Omron Sysmac Studio project distributing_station_with_timer_1.9_no_erorcheck (1) (Sysmac Studio 1.54.0.64019, StandardProject)

# Controller new_Controller_0: NJ301-1100 version 1.14
Units and slaves: Node1 : NX-ECC201 (E001); Unit 1 : NX-PC0020 (N1); Unit 2 : NX-ID5442 (N2); Unit 3 : NX-PC0010 (N3); Unit 4 : NX-PC0020 (N4); Unit 5 : NX-OD5121 (N5); Unit 6 : NX-PC0010 (N6); Power Supply : NJ-Px3001; CPU : NJ301-1100; 0 [Unit 0] : CJ1W-AD041-V1 (J01); 1 [Unit 1] : CJ1W-DA041 (J02); 2 : CJ1W-ID211 (J03); 3 : CJ1W-OC211 (J04)
Task PrimaryTask (priority 4, period or condition 1000): Program0

VAR_GLOBAL
    Station_1B2 : BOOL;  (* Ejection Cylinder Extended; at IOBus://rack#0/slot#2/Ch1_In/Ch1_In01; published *)
    Station_1B1 : BOOL;  (* Ejection Cylinder retracted; at IOBus://rack#0/slot#2/Ch1_In/Ch1_In02; published *)
    Station_2B1 : BOOL;  (* Workpiece gripped; at IOBus://rack#0/slot#2/Ch1_In/Ch1_In03; published *)
    Station_3S1 : BOOL;  (* arm_in_magazine; at IOBus://rack#0/slot#2/Ch1_In/Ch1_In04; published *)
    Station_3S2 : BOOL;  (* arm_in_downstream; at IOBus://rack#0/slot#2/Ch1_In/Ch1_In05; published *)
    Station_B4 : BOOL;  (* Magzine empty; at IOBus://rack#0/slot#2/Ch1_In/Ch1_In06; published *)
    Panel_S1 : BOOL;  (* start_button; at IOBus://rack#0/slot#2/Ch1_In/Ch1_In08; published *)
    Panel_S2 : BOOL;  (* stop_button; at IOBus://rack#0/slot#2/Ch1_In/Ch1_In09; published *)
    Panel_S4 : BOOL;  (* reset_button; at IOBus://rack#0/slot#2/Ch1_In/Ch1_In11; published *)
    Station_1Y1 : BOOL;  (* Magzine eject; at IOBus://rack#0/slot#3/Ch1_Out/Ch1_Out00; published *)
    Station_2Y1 : BOOL;  (* Vacuum on; at IOBus://rack#0/slot#3/Ch1_Out/Ch1_Out01; published *)
    Station_2Y2 : BOOL;  (* Ejector_Pulse_On; at IOBus://rack#0/slot#3/Ch1_Out/Ch1_Out02; published *)
    Station_3Y1 : BOOL;  (* arm_2_magazine; at IOBus://rack#0/slot#3/Ch1_Out/Ch1_Out03; published *)
    Station_3Y2 : BOOL;  (* arm_2_downstream; at IOBus://rack#0/slot#3/Ch1_Out/Ch1_Out04; published *)
    Station_H1 : BOOL;  (* start light; at IOBus://rack#0/slot#3/Ch1_Out/Ch1_Out08; published *)
    Station_H2 : BOOL;  (* reset light; at IOBus://rack#0/slot#3/Ch1_Out/Ch1_Out09; published *)
    Panel_H3 : BOOL;  (* Q1 light; at IOBus://rack#0/slot#3/Ch1_Out/Ch1_Out10; published *)
    Panel_H4 : BOOL;  (* Q2 light; at IOBus://rack#0/slot#3/Ch1_Out/Ch1_Out11; published *)
END_VAR

PROGRAM Program0
VAR
    FB_Panel_Distribution : FB_Panel;
    run_mode : BOOL;
    start_light : BOOL;
    reset_light : BOOL;
    pause_mode : BOOL;
    reset_mode : BOOL;
    T1_error_environment : BOOL;  (* t1 arm error *)
    error_mode : BOOL;
    T2_error_environment : BOOL;  (* t2 ejector error *)
    T1_to_end : BOOL;
    T1_to_home : BOOL;
    T1_at_home : BOOL;
    T1_at_end : BOOL;
    T2_to_end : BOOL;
    T2_to_home : BOOL;
    T2_at_home : BOOL;
    T2_at_end : BOOL;
    T2_Actuator_Env : T2_Actuator_No_RS_Controllable;
    T1_Actuator_Env : T1_Actuator_Controllable;
    Distrabution_Station_Logic_Env : Distrabuting_Station_Logic;
    manual_mode : BOOL;  (* empty boolean to control manual mode *)
    Dis_Logic_reset_light : BOOL;
    Dis_Logic_start_light : BOOL;
    Dis_Logic_empty_mag_light : BOOL;
    arm_to_end : BOOL;
    arm_to_home : BOOL;
    Dis_Logic_arm_to_end : BOOL;
    Dis_Logic_arm_to_home : BOOL;
    Dis_Logic_extend_mag_slide : BOOL;
    Dis_Logic_retract_mag_slide : BOOL;
END_VAR
VAR_EXTERNAL
    Station_3S1 : BOOL;
    Panel_S2 : BOOL;
    Station_3Y2 : BOOL;
    Station_3S2 : BOOL;
    Panel_S1 : BOOL;
    Station_3Y1 : BOOL;
    Station_H1 : BOOL;
    Station_H2 : BOOL;
    Panel_S4 : BOOL;
    Panel_H4 : BOOL;
    Station_1B1 : BOOL;
    Station_1B2 : BOOL;
    Station_1Y1 : BOOL;
    Station_2B1 : BOOL;
    Station_B4 : BOOL;
    Station_2Y1 : BOOL;
    Station_2Y2 : BOOL;
END_VAR

(* Section Section0: ladder, written here as Structured Text *)

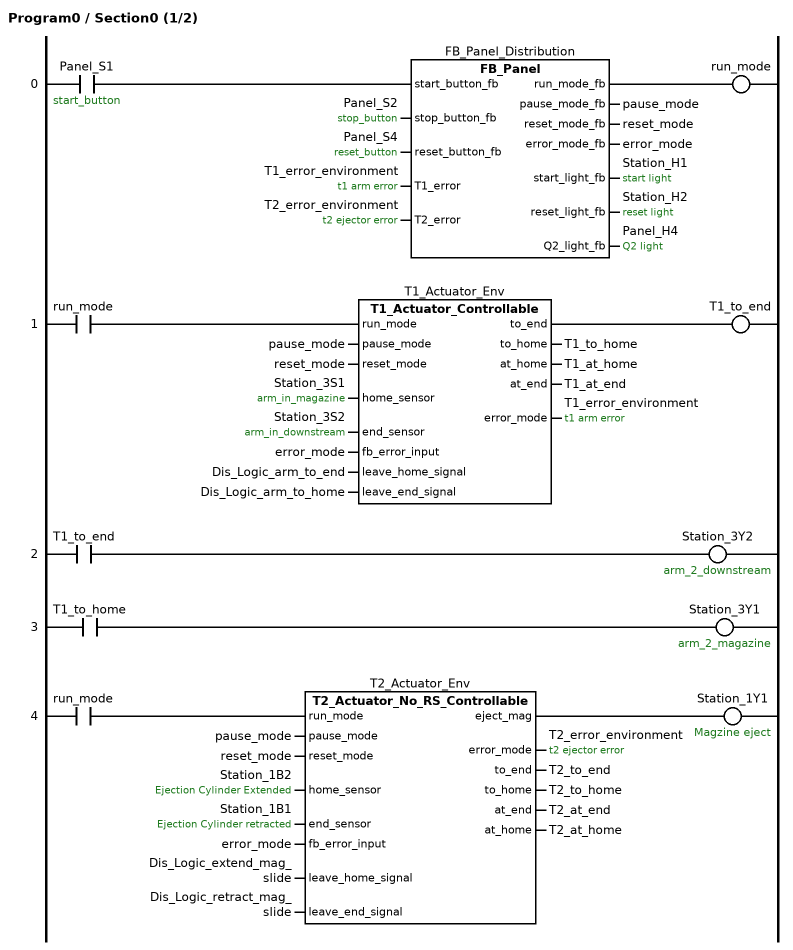
(* Rung 0 *)
FB_Panel_Distribution(start_button_fb := Panel_S1, stop_button_fb := Panel_S2, reset_button_fb := Panel_S4, T1_error := T1_error_environment, T2_error := T2_error_environment, pause_mode_fb => pause_mode, reset_mode_fb => reset_mode, error_mode_fb => error_mode, start_light_fb => Station_H1, reset_light_fb => Station_H2, Q2_light_fb => Panel_H4);
run_mode := FB_Panel_Distribution.run_mode_fb;
(* Rung 1 *)
T1_Actuator_Env(run_mode := run_mode, pause_mode := pause_mode, reset_mode := reset_mode, home_sensor := Station_3S1, end_sensor := Station_3S2, fb_error_input := error_mode, leave_home_signal := Dis_Logic_arm_to_end, leave_end_signal := Dis_Logic_arm_to_home, to_home => T1_to_home, at_home => T1_at_home, at_end => T1_at_end, error_mode => T1_error_environment);
T1_to_end := T1_Actuator_Env.to_end;
(* Rung 2 *)
Station_3Y2 := T1_to_end;
(* Rung 3 *)
Station_3Y1 := T1_to_home;
(* Rung 4 *)
T2_Actuator_Env(run_mode := run_mode, pause_mode := pause_mode, reset_mode := reset_mode, home_sensor := Station_1B2, end_sensor := Station_1B1, fb_error_input := error_mode, leave_home_signal := Dis_Logic_extend_mag_slide, leave_end_signal := Dis_Logic_retract_mag_slide, error_mode => T2_error_environment, to_end => T2_to_end, to_home => T2_to_home, at_end => T2_at_end, at_home => T2_at_home);
Station_1Y1 := T2_Actuator_Env.eject_mag;

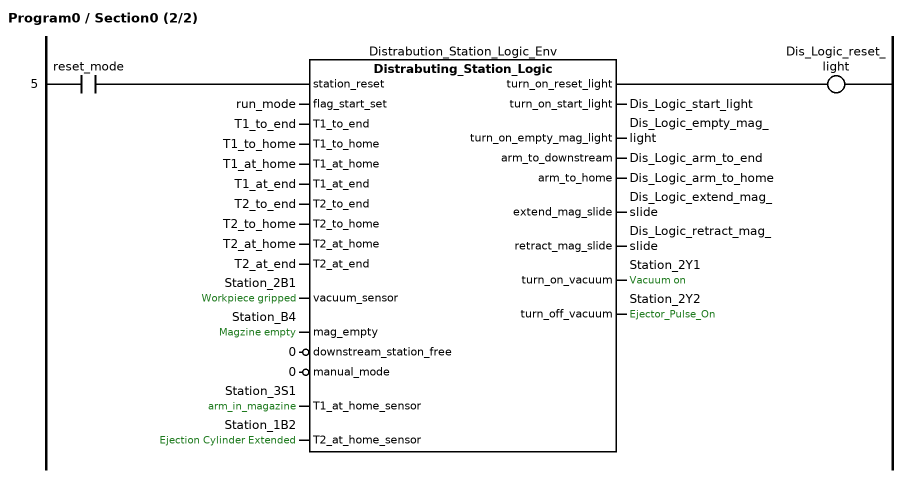
(* Rung 5 *)
Distrabution_Station_Logic_Env(station_reset := reset_mode, flag_start_set := run_mode, T1_to_end := T1_to_end, T1_to_home := T1_to_home, T1_at_home := T1_at_home, T1_at_end := T1_at_end, T2_to_end := T2_to_end, T2_to_home := T2_to_home, T2_at_home := T2_at_home, T2_at_end := T2_at_end, vacuum_sensor := Station_2B1, mag_empty := Station_B4, downstream_station_free := NOT 0, manual_mode := NOT 0, T1_at_home_sensor := Station_3S1, T2_at_home_sensor := Station_1B2, turn_on_start_light => Dis_Logic_start_light, turn_on_empty_mag_light => Dis_Logic_empty_mag_light, arm_to_downstream => Dis_Logic_arm_to_end, arm_to_home => Dis_Logic_arm_to_home, extend_mag_slide => Dis_Logic_extend_mag_slide, retract_mag_slide => Dis_Logic_retract_mag_slide, turn_on_vacuum => Station_2Y1, turn_off_vacuum => Station_2Y2);
Dis_Logic_reset_light := Distrabution_Station_Logic_Env.turn_on_reset_light;
END_PROGRAM

FUNCTION_BLOCK FB_Panel
VAR
    RS_run_mode : RS;
    RS_reset_mode : RS;
    RS_run_mode_reset : BOOL;  (* reset run mode RS *)
END_VAR
VAR_OUTPUT
    run_mode_fb : BOOL;
    pause_mode_fb : BOOL;
    reset_mode_fb : BOOL;
    error_mode_fb : BOOL;
END_VAR
VAR_INPUT
    start_button_fb : BOOL;
    stop_button_fb : BOOL;
    reset_button_fb : BOOL;
    T1_error : BOOL;  (* arm error mode input *)
    T2_error : BOOL;  (* ejector cylinder error mode input *)
END_VAR
VAR_OUTPUT
    start_light_fb : BOOL;
    reset_light_fb : BOOL;
    Q2_light_fb : BOOL;
END_VAR
(* ladder, written here as Structured Text *)

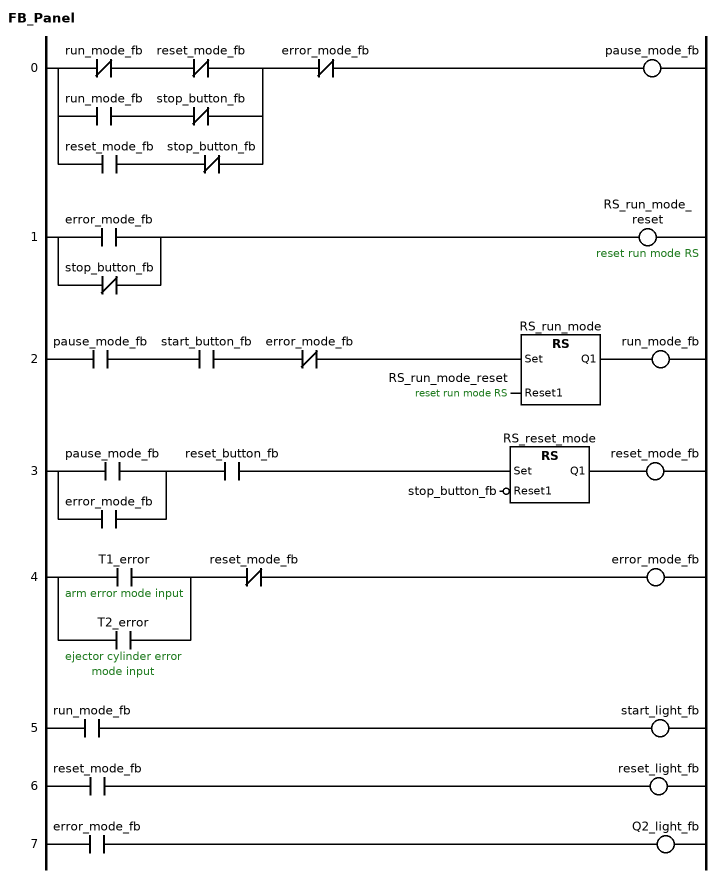
(* Rung 0 *)
pause_mode_fb := ((NOT run_mode_fb AND NOT reset_mode_fb) OR (run_mode_fb AND NOT stop_button_fb) OR (reset_mode_fb AND NOT stop_button_fb)) AND NOT error_mode_fb;
(* Rung 1 *)
RS_run_mode_reset := error_mode_fb OR NOT stop_button_fb;
(* Rung 2 *)
RS_run_mode(Set := pause_mode_fb AND start_button_fb AND NOT error_mode_fb, Reset1 := RS_run_mode_reset);
run_mode_fb := RS_run_mode.Q1;
(* Rung 3 *)
RS_reset_mode(Set := (pause_mode_fb OR error_mode_fb) AND reset_button_fb, Reset1 := NOT stop_button_fb);
reset_mode_fb := RS_reset_mode.Q1;
(* Rung 4 *)
error_mode_fb := (T1_error OR T2_error) AND NOT reset_mode_fb;
(* Rung 5 *)
start_light_fb := run_mode_fb;
(* Rung 6 *)
reset_light_fb := reset_mode_fb;
(* Rung 7 *)
Q2_light_fb := error_mode_fb;
END_FUNCTION_BLOCK

FUNCTION_BLOCK T1_Actuator_Controllable
VAR
    to_end_RS : RS;
    at_home_RS : RS;
    at_end_RS : RS;
    to_home_RS : RS;
    reset_to_end_RS : BOOL;  (* reset to end RS *)
    reset_at_end_RS : BOOL;  (* reset at end RS *)
    reset_to_home_RS : BOOL;  (* reset to home RS signal *)
    reset_at_home_RS : BOOL;  (* reset at home RS *)
    initialise_station : BOOL;  (* initialise station to at home state *)
    to_end_pause : BOOL;  (* pause state from to end state *)
    to_home_pause : BOOL;  (* pause state from to home state *)
    run : BOOL;
    insitilise_station_RS : RS;
    to_end_pause_RS : RS;
    reset_to_end_pause_RS : BOOL;  (* reset to end pause RS *)
    to_home_pause_RS : RS;
    reset_to_home_pause_RS : BOOL;  (* reset to home pause RS *)
    exiting_to_home_pause_RS : RS;
    exiting_to_home_pause : BOOL;  (* exiting to home pause mode *)
    exiting_to_end_pause : BOOL;  (* exiting to end pause mode *)
    exiting_to_end_pause_RS : RS;
    T1_reset_mode : BOOL;  (* arm reset mode *)
    T1_reset_mode_RS : RS;
    reset_T1_reset_mode_RS : BOOL;  (* reset T1 reset mode RS *)
    initialise_complete : BOOL;  (* On when start up initilisation is complete *)
    initialise_complete_RS : RS;
    error_mode_timer : AccumulationTimer;
    ErrorTimeET : TIME;
    error_mode_timer_reset : BOOL;  (* resets error mode's accumulation timer to 0 *)
    entering_to_home_pause_RS : RS;
    entering_to_home_pause : BOOL;
END_VAR
VAR_INPUT
    run_mode : BOOL;  (* run mode *)
    pause_mode : BOOL;  (* pause mode *)
    reset_mode : BOOL;  (* reset mode *)
    home_sensor : BOOL;  (* sensor at home position *)
    end_sensor : BOOL;  (* sensor at end position *)
    fb_error_input : BOOL;  (* FB panel error input (Other Station Error) *)
    leave_home_signal : BOOL;  (* external signal to leave home position *)
    leave_end_signal : BOOL;  (* external signal to leave end position *)
END_VAR
VAR_OUTPUT
    to_end : BOOL;  (* going to end position *)
    to_home : BOOL;  (* going to home position *)
    at_home : BOOL;  (* at home position *)
    at_end : BOOL;  (* at end position *)
    error_mode : BOOL;  (* error mode for when arm does not reach desination in allocated time or error occurs in other stations *)
END_VAR
(* ladder, written here as Structured Text *)

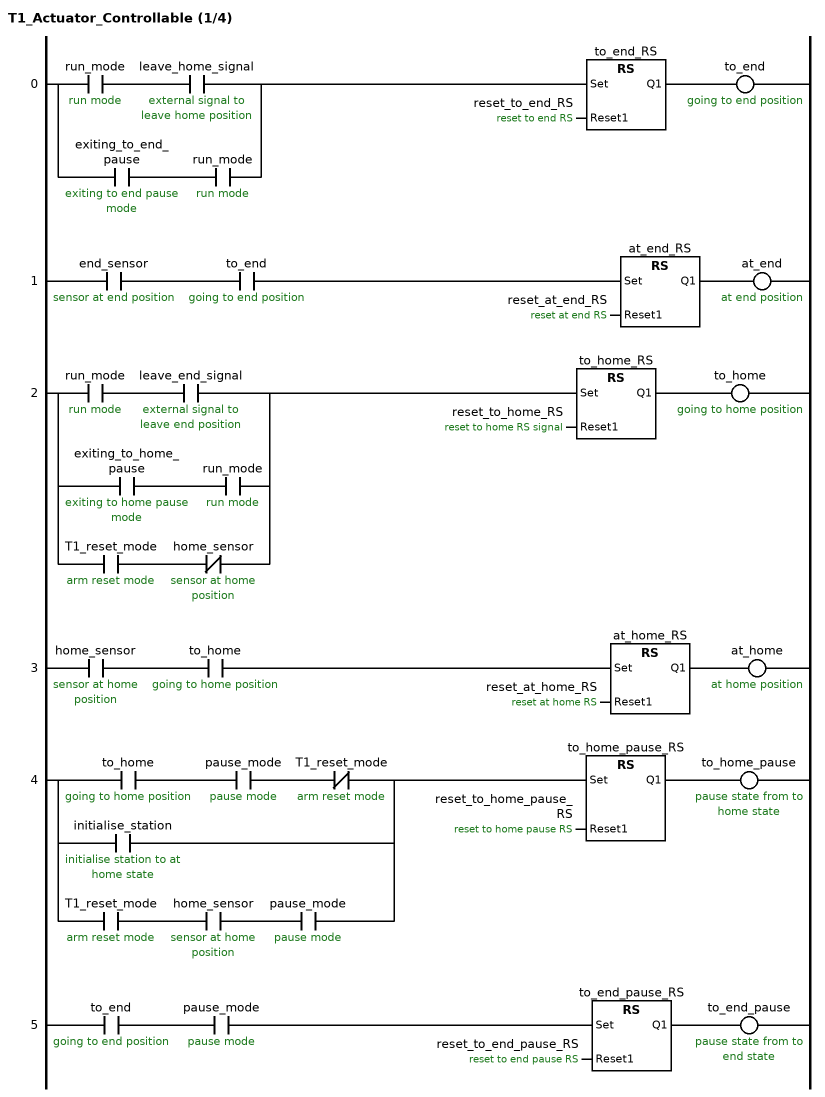
(* Rung 0 *)
to_end_RS(Set := (run_mode AND leave_home_signal) OR (exiting_to_end_pause AND run_mode), Reset1 := reset_to_end_RS);
to_end := to_end_RS.Q1;
(* Rung 1 *)
at_end_RS(Set := end_sensor AND to_end, Reset1 := reset_at_end_RS);
at_end := at_end_RS.Q1;
(* Rung 2 *)
to_home_RS(Set := (run_mode AND leave_end_signal) OR (exiting_to_home_pause AND run_mode) OR (T1_reset_mode AND NOT home_sensor), Reset1 := reset_to_home_RS);
to_home := to_home_RS.Q1;
(* Rung 3 *)
at_home_RS(Set := home_sensor AND to_home, Reset1 := reset_at_home_RS);
at_home := at_home_RS.Q1;
(* Rung 4 *)
to_home_pause_RS(Set := (to_home AND pause_mode AND NOT T1_reset_mode) OR initialise_station OR (T1_reset_mode AND home_sensor AND pause_mode), Reset1 := reset_to_home_pause_RS);
to_home_pause := to_home_pause_RS.Q1;
(* Rung 5 *)
to_end_pause_RS(Set := to_end AND pause_mode, Reset1 := reset_to_end_pause_RS);
to_end_pause := to_end_pause_RS.Q1;

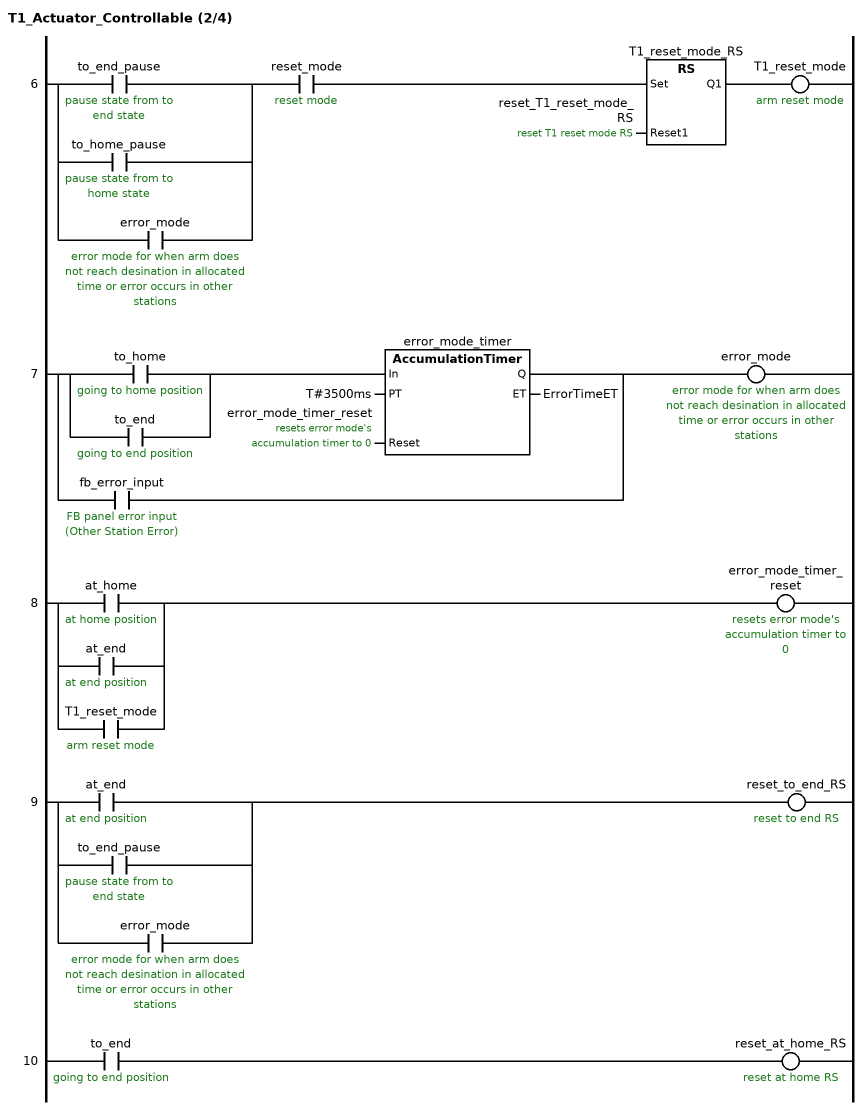
(* Rung 6 *)
T1_reset_mode_RS(Set := (to_end_pause OR to_home_pause OR error_mode) AND reset_mode, Reset1 := reset_T1_reset_mode_RS);
T1_reset_mode := T1_reset_mode_RS.Q1;
(* Rung 7 *)
error_mode_timer(In := to_home OR to_end, PT := T#3500ms, Reset := error_mode_timer_reset, ET => ErrorTimeET);
error_mode := error_mode_timer.Q OR fb_error_input;
(* Rung 8 *)
error_mode_timer_reset := at_home OR at_end OR T1_reset_mode;
(* Rung 9 *)
reset_to_end_RS := at_end OR to_end_pause OR error_mode;
(* Rung 10 *)
reset_at_home_RS := to_end;

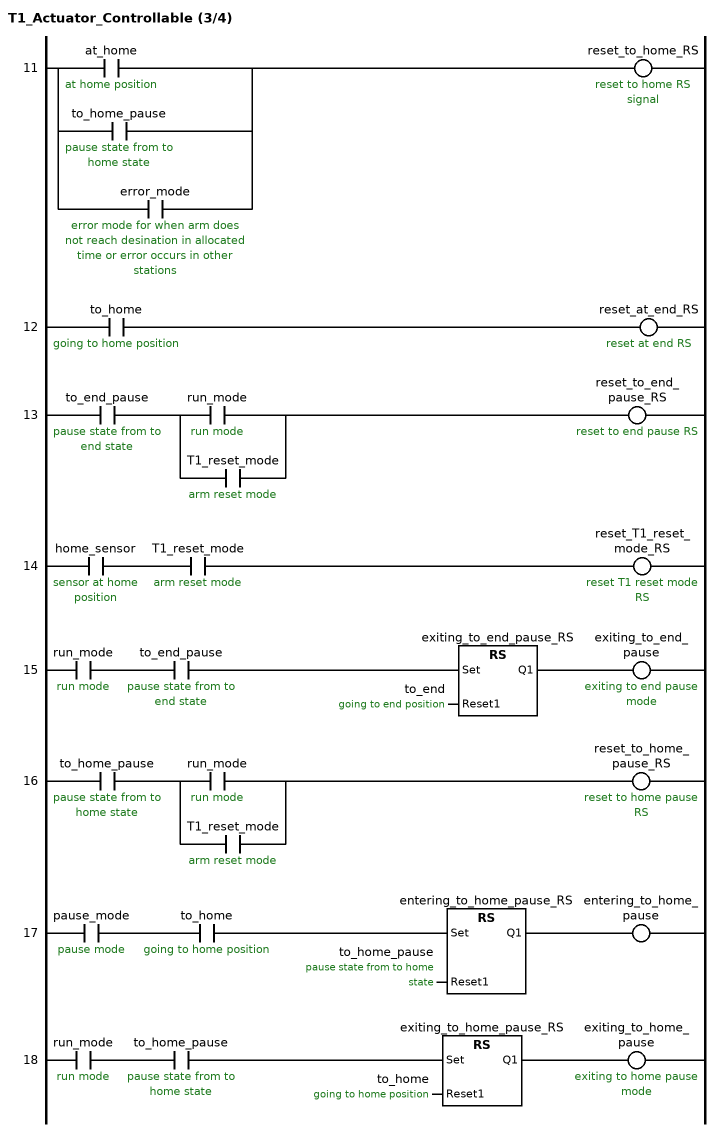
(* Rung 11 *)
reset_to_home_RS := at_home OR to_home_pause OR error_mode;
(* Rung 12 *)
reset_at_end_RS := to_home;
(* Rung 13 *)
reset_to_end_pause_RS := to_end_pause AND (run_mode OR T1_reset_mode);
(* Rung 14 *)
reset_T1_reset_mode_RS := home_sensor AND T1_reset_mode;
(* Rung 15 *)
exiting_to_end_pause_RS(Set := run_mode AND to_end_pause, Reset1 := to_end);
exiting_to_end_pause := exiting_to_end_pause_RS.Q1;
(* Rung 16 *)
reset_to_home_pause_RS := to_home_pause AND (run_mode OR T1_reset_mode);
(* Rung 17 *)
entering_to_home_pause_RS(Set := pause_mode AND to_home, Reset1 := to_home_pause);
entering_to_home_pause := entering_to_home_pause_RS.Q1;
(* Rung 18 *)
exiting_to_home_pause_RS(Set := run_mode AND to_home_pause, Reset1 := to_home);
exiting_to_home_pause := exiting_to_home_pause_RS.Q1;

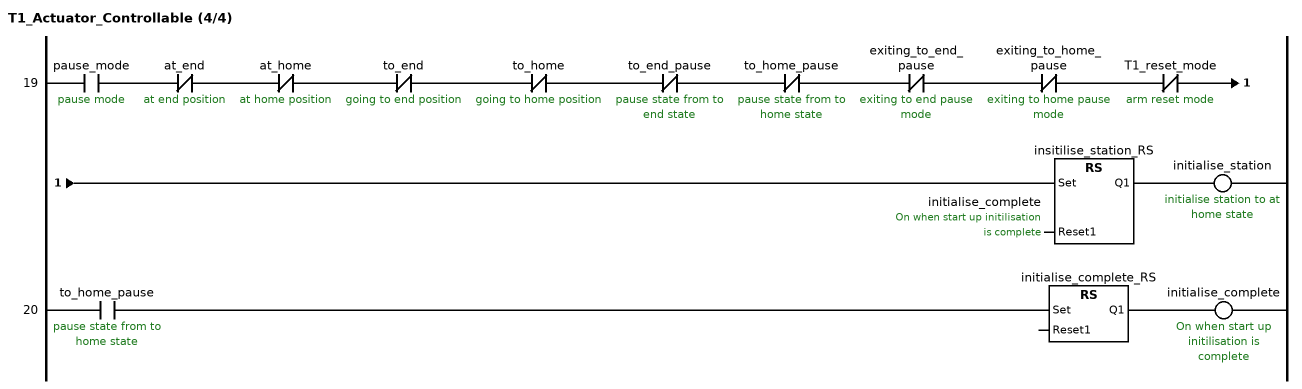
(* Rung 19 *)
insitilise_station_RS(Set := pause_mode AND NOT at_end AND NOT at_home AND NOT to_end AND NOT to_home AND NOT to_end_pause AND NOT to_home_pause AND NOT exiting_to_end_pause AND NOT exiting_to_home_pause AND NOT T1_reset_mode, Reset1 := initialise_complete);
initialise_station := insitilise_station_RS.Q1;
(* Rung 20 *)
initialise_complete_RS(Set := to_home_pause);
initialise_complete := initialise_complete_RS.Q1;
END_FUNCTION_BLOCK

FUNCTION_BLOCK T2_Actuator
VAR
    to_end_RS : RS;
    at_end_RS : RS;
    to_home_RS : RS;
    at_home_RS : RS;
    reset_to_end_RS : BOOL;
    reset_at_end_RS : BOOL;
    reset_to_home_RS : BOOL;
    reset_at_home_RS : BOOL;
    T2_reset_mode : BOOL;  (* T2 reset mode *)
    T2_reset_mode_RS : RS;
    reset_T2_reset_mode_RS : BOOL;
END_VAR
VAR_INPUT
    run_mode : BOOL;
    pause_mode : BOOL;
    reset_mode : BOOL;
    home_sensor : BOOL;
    end_sensor : BOOL;
END_VAR
VAR_OUTPUT
    to_end : BOOL;
    to_home : BOOL;
    at_end : BOOL;
    at_home : BOOL;
END_VAR
(* ladder, written here as Structured Text *)

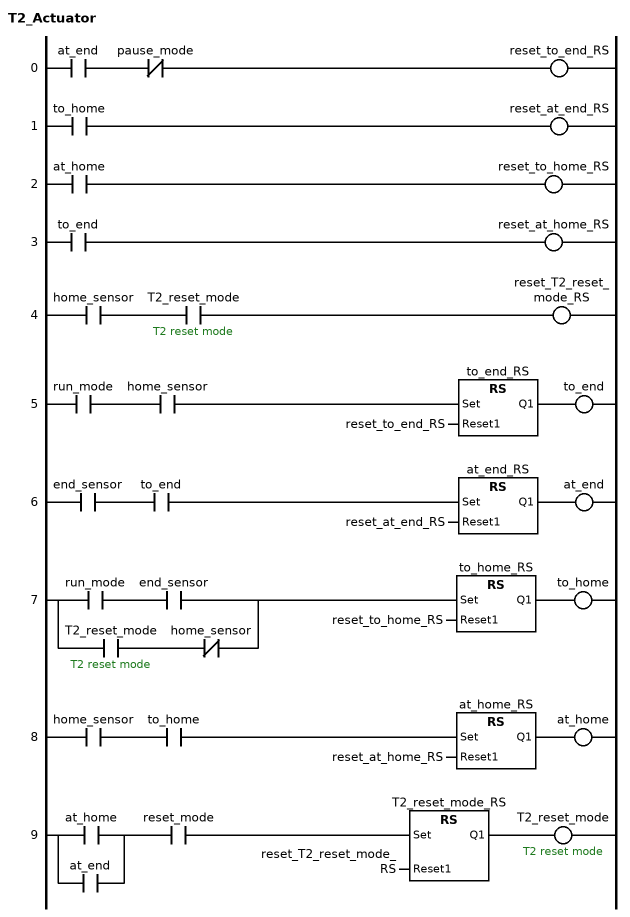
(* Rung 0 *)
reset_to_end_RS := at_end AND NOT pause_mode;
(* Rung 1 *)
reset_at_end_RS := to_home;
(* Rung 2 *)
reset_to_home_RS := at_home;
(* Rung 3 *)
reset_at_home_RS := to_end;
(* Rung 4 *)
reset_T2_reset_mode_RS := home_sensor AND T2_reset_mode;
(* Rung 5 *)
to_end_RS(Set := run_mode AND home_sensor, Reset1 := reset_to_end_RS);
to_end := to_end_RS.Q1;
(* Rung 6 *)
at_end_RS(Set := end_sensor AND to_end, Reset1 := reset_at_end_RS);
at_end := at_end_RS.Q1;
(* Rung 7 *)
to_home_RS(Set := (run_mode AND end_sensor) OR (T2_reset_mode AND NOT home_sensor), Reset1 := reset_to_home_RS);
to_home := to_home_RS.Q1;
(* Rung 8 *)
at_home_RS(Set := home_sensor AND to_home, Reset1 := reset_at_home_RS);
at_home := at_home_RS.Q1;
(* Rung 9 *)
T2_reset_mode_RS(Set := (at_home OR at_end) AND reset_mode, Reset1 := reset_T2_reset_mode_RS);
T2_reset_mode := T2_reset_mode_RS.Q1;
END_FUNCTION_BLOCK

FUNCTION_BLOCK T2_Actuator_No_RS_Controllable
VAR
    T2_reset_mode : BOOL;  (* T2 reset mode *)
    error_mode_timer : AccumulationTimer;
    error_mode_timer_reset : BOOL;
    ErrorTimeET : TIME;
END_VAR
VAR_INPUT
    run_mode : BOOL;
    pause_mode : BOOL;
    reset_mode : BOOL;
    home_sensor : BOOL;
    end_sensor : BOOL;
    fb_error_input : BOOL;
    leave_home_signal : BOOL;  (* External signal to leave home position *)
    leave_end_signal : BOOL;  (* Exernal signal to leave end position *)
END_VAR
VAR_OUTPUT
    eject_mag : BOOL;
    error_mode : BOOL;
    to_end : BOOL;
    to_home : BOOL;
    at_end : BOOL;
    at_home : BOOL;
END_VAR
(* ladder, written here as Structured Text *)

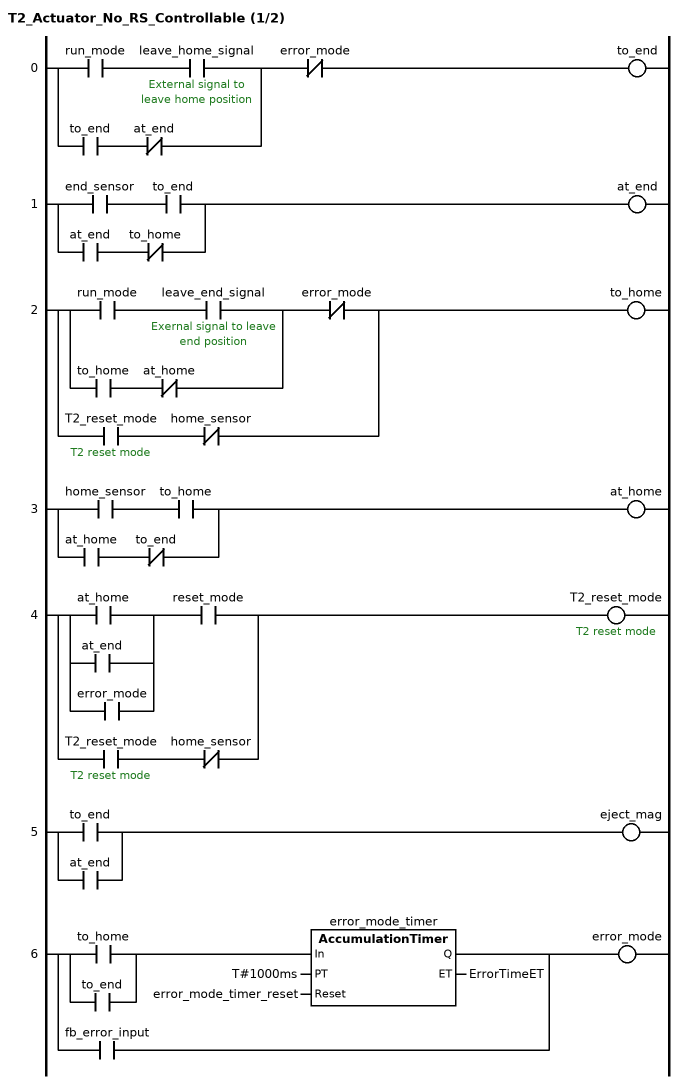
(* Rung 0 *)
to_end := ((run_mode AND leave_home_signal) OR (to_end AND NOT at_end)) AND NOT error_mode;
(* Rung 1 *)
at_end := (end_sensor AND to_end) OR (at_end AND NOT to_home);
(* Rung 2 *)
to_home := (((run_mode AND leave_end_signal) OR (to_home AND NOT at_home)) AND NOT error_mode) OR (T2_reset_mode AND NOT home_sensor);
(* Rung 3 *)
at_home := (home_sensor AND to_home) OR (at_home AND NOT to_end);
(* Rung 4 *)
T2_reset_mode := ((at_home OR at_end OR error_mode) AND reset_mode) OR (T2_reset_mode AND NOT home_sensor);
(* Rung 5 *)
eject_mag := to_end OR at_end;
(* Rung 6 *)
error_mode_timer(In := to_home OR to_end, PT := T#1000ms, Reset := error_mode_timer_reset, ET => ErrorTimeET);
error_mode := error_mode_timer.Q OR fb_error_input;

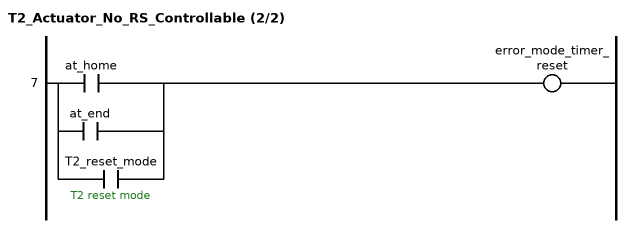
(* Rung 7 *)
error_mode_timer_reset := at_home OR at_end OR T2_reset_mode;
END_FUNCTION_BLOCK

FUNCTION_BLOCK Distrabuting_Station_Logic
VAR
    cycle_start : BOOL;  (* start of station cycle *)
    reset_light : BOOL;
    moving_to_initial_pos : BOOL;
    station_initial_pos : BOOL;
    set_reset_flag_off : BOOL;
    is_downstream_station_free : BOOL;
    mag_status : BOOL;
    empty_mag_error_solved : BOOL;  (* empty mag is solved and start button is pressed *)
    set_cycle_end_on : BOOL;
    loop_to_cycle_start : BOOL;
    loop_to_mag_status : BOOL;
    initialise_reset : RS;
    initialised_station : BOOL;  (* variable to allow station to initialise on reset mode once *)
    arm_to_downstream_cycle_1 : BOOL;
    arm_to_downstream_cycle_2 : BOOL;
    arm_to_home_cycle_1 : BOOL;
    arm_to_home_cycle_2 : BOOL;
    turn_on_start_light_cycle_1 : BOOL;
    turn_on_start_light_cycle_2 : BOOL;
    retract_mag_slide_cycle_1 : BOOL;
    retract_mag_slide_cycle_2 : BOOL;
    piece_ejected : BOOL;
END_VAR
VAR_INPUT
    station_reset : BOOL;
    flag_start_set : BOOL;
    T1_to_end : BOOL;
    T1_to_home : BOOL;
    T1_at_home : BOOL;
    T1_at_end : BOOL;
    T2_to_end : BOOL;
    T2_to_home : BOOL;
    T2_at_home : BOOL;
    T2_at_end : BOOL;
    vacuum_sensor : BOOL;
    mag_empty : BOOL;
    downstream_station_free : BOOL;
    manual_mode : BOOL;
    T1_at_home_sensor : BOOL;
    T2_at_home_sensor : BOOL;
END_VAR
VAR_OUTPUT
    turn_on_reset_light : BOOL;
    turn_on_start_light : BOOL;
    turn_on_empty_mag_light : BOOL;
    arm_to_downstream : BOOL;
    arm_to_home : BOOL;
    extend_mag_slide : BOOL;
    retract_mag_slide : BOOL;
    turn_on_vacuum : BOOL;
    turn_off_vacuum : BOOL;
END_VAR
VAR
    _p1 : BOOL;
    _p2 : BOOL;
    _p3 : BOOL;
    _p4 : BOOL;
END_VAR
(* ladder, written here as Structured Text *)

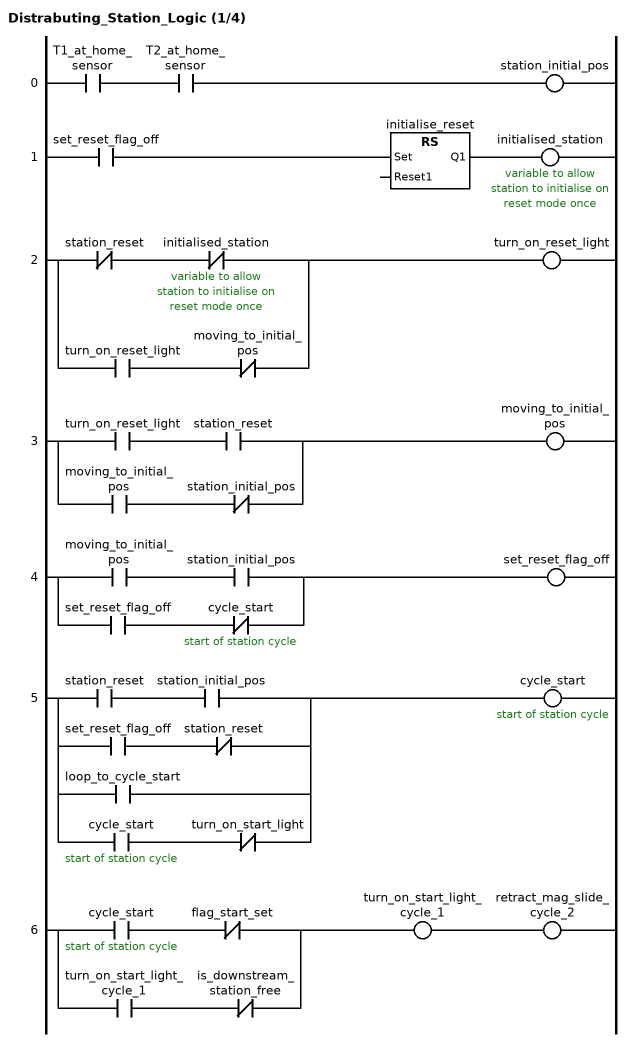
(* Rung 0 *)
station_initial_pos := T1_at_home_sensor AND T2_at_home_sensor;
(* Rung 1 *)
initialise_reset(Set := set_reset_flag_off);
initialised_station := initialise_reset.Q1;
(* Rung 2 *)
turn_on_reset_light := (NOT station_reset AND NOT initialised_station) OR (turn_on_reset_light AND NOT moving_to_initial_pos);
(* Rung 3 *)
moving_to_initial_pos := (turn_on_reset_light AND station_reset) OR (moving_to_initial_pos AND NOT station_initial_pos);
(* Rung 4 *)
set_reset_flag_off := (moving_to_initial_pos AND station_initial_pos) OR (set_reset_flag_off AND NOT cycle_start);
(* Rung 5 *)
cycle_start := (station_reset AND station_initial_pos) OR (set_reset_flag_off AND NOT station_reset) OR loop_to_cycle_start OR (cycle_start AND NOT turn_on_start_light);
(* Rung 6 *)
_p1 := (cycle_start AND NOT flag_start_set) OR (turn_on_start_light_cycle_1 AND NOT is_downstream_station_free);
turn_on_start_light_cycle_1 := _p1;
retract_mag_slide_cycle_2 := _p1;

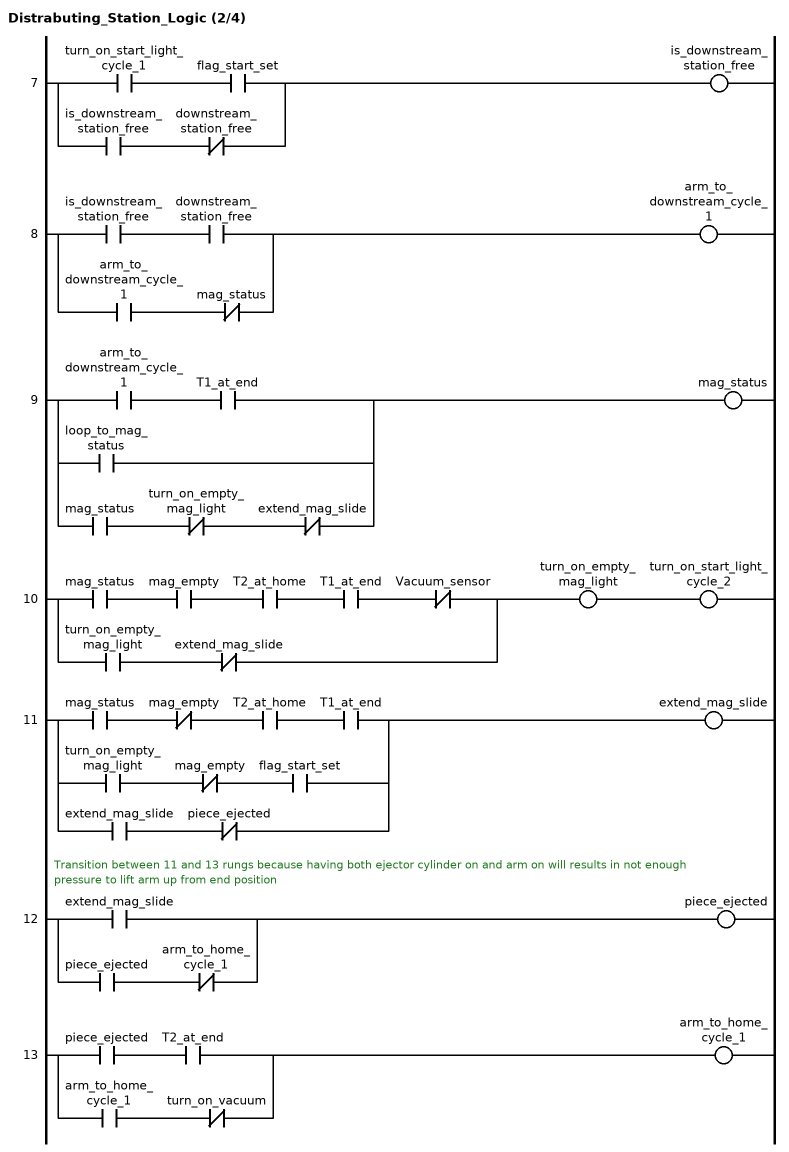
(* Rung 7 *)
is_downstream_station_free := (turn_on_start_light_cycle_1 AND flag_start_set) OR (is_downstream_station_free AND NOT downstream_station_free);
(* Rung 8 *)
arm_to_downstream_cycle_1 := (is_downstream_station_free AND downstream_station_free) OR (arm_to_downstream_cycle_1 AND NOT mag_status);
(* Rung 9 *)
mag_status := (arm_to_downstream_cycle_1 AND T1_at_end) OR loop_to_mag_status OR (mag_status AND NOT turn_on_empty_mag_light AND NOT extend_mag_slide);
(* Rung 10 *)
_p2 := (mag_status AND mag_empty AND T2_at_home AND T1_at_end AND NOT Vacuum_sensor) OR (turn_on_empty_mag_light AND NOT extend_mag_slide);
turn_on_empty_mag_light := _p2;
turn_on_start_light_cycle_2 := _p2;
(* Rung 11 *)
extend_mag_slide := (mag_status AND NOT mag_empty AND T2_at_home AND T1_at_end) OR (turn_on_empty_mag_light AND NOT mag_empty AND flag_start_set) OR (extend_mag_slide AND NOT piece_ejected);
(* Rung 12: Transition between 11 and 13 rungs because having both ejector cylinder on and arm on will results in not enough pressure to lift arm up from end position *)
piece_ejected := extend_mag_slide OR (piece_ejected AND NOT arm_to_home_cycle_1);
(* Rung 13 *)
arm_to_home_cycle_1 := (piece_ejected AND T2_at_end) OR (arm_to_home_cycle_1 AND NOT turn_on_vacuum);

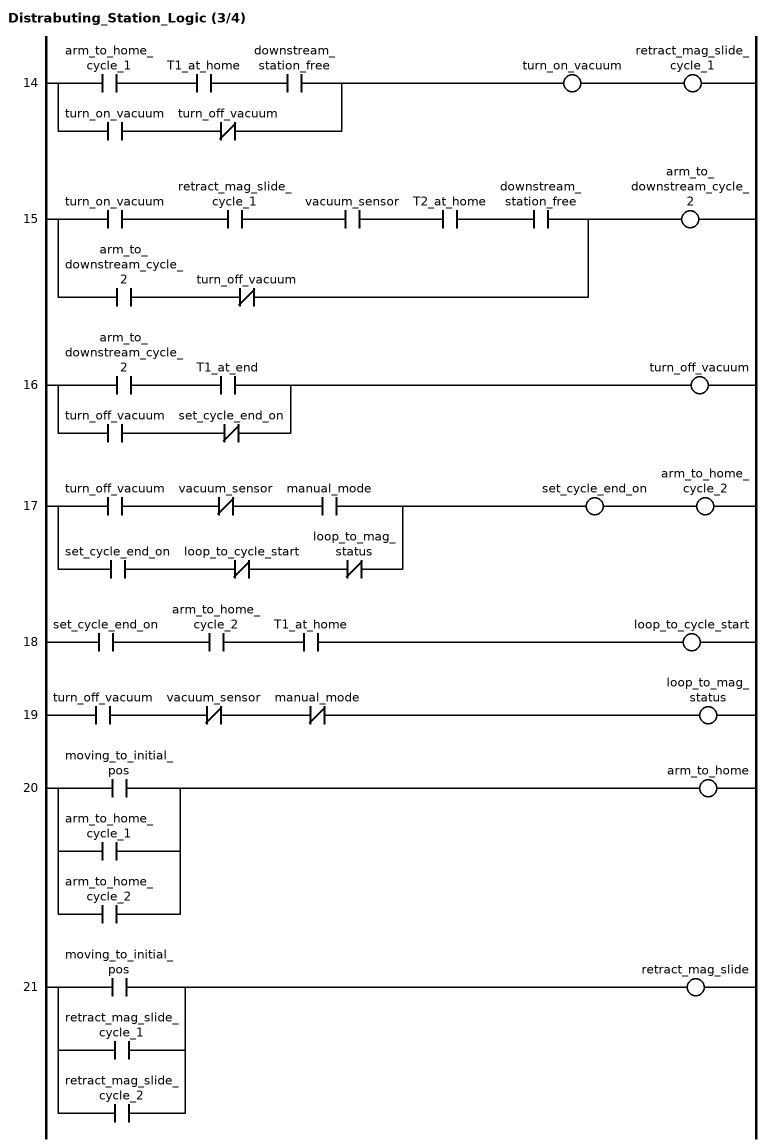
(* Rung 14 *)
_p3 := (arm_to_home_cycle_1 AND T1_at_home AND downstream_station_free) OR (turn_on_vacuum AND NOT turn_off_vacuum);
turn_on_vacuum := _p3;
retract_mag_slide_cycle_1 := _p3;
(* Rung 15 *)
arm_to_downstream_cycle_2 := (turn_on_vacuum AND retract_mag_slide_cycle_1 AND vacuum_sensor AND T2_at_home AND downstream_station_free) OR (arm_to_downstream_cycle_2 AND NOT turn_off_vacuum);
(* Rung 16 *)
turn_off_vacuum := (arm_to_downstream_cycle_2 AND T1_at_end) OR (turn_off_vacuum AND NOT set_cycle_end_on);
(* Rung 17 *)
_p4 := (turn_off_vacuum AND NOT vacuum_sensor AND manual_mode) OR (set_cycle_end_on AND NOT loop_to_cycle_start AND NOT loop_to_mag_status);
set_cycle_end_on := _p4;
arm_to_home_cycle_2 := _p4;
(* Rung 18 *)
loop_to_cycle_start := set_cycle_end_on AND arm_to_home_cycle_2 AND T1_at_home;
(* Rung 19 *)
loop_to_mag_status := turn_off_vacuum AND NOT vacuum_sensor AND NOT manual_mode;
(* Rung 20 *)
arm_to_home := moving_to_initial_pos OR arm_to_home_cycle_1 OR arm_to_home_cycle_2;
(* Rung 21 *)
retract_mag_slide := moving_to_initial_pos OR retract_mag_slide_cycle_1 OR retract_mag_slide_cycle_2;

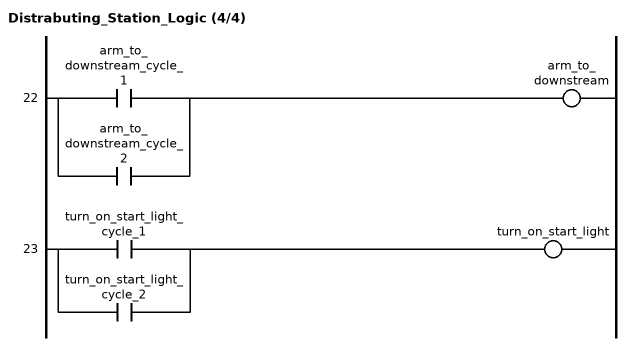
(* Rung 22 *)
arm_to_downstream := arm_to_downstream_cycle_1 OR arm_to_downstream_cycle_2;
(* Rung 23 *)
turn_on_start_light := turn_on_start_light_cycle_1 OR turn_on_start_light_cycle_2;
END_FUNCTION_BLOCK

FUNCTION_BLOCK Copy_1_of_Distrabuting_Station_Logic
VAR
    cycle_start : BOOL;  (* start of station cycle *)
    reset_light : BOOL;
    turn_on_reset_light : BOOL;
    moving_to_initial_pos : BOOL;
    station_initial_pos : BOOL;
    set_reset_flag_off : BOOL;
    reset_flag_set_off : BOOL;
    station_reset : BOOL;
    flag_start_set : BOOL;
    turn_on_start_light : BOOL;
    is_downstream_station_free : BOOL;
    downstream_station_free : BOOL;
    arm_to_downstream : BOOL;
    mag_status : BOOL;
    turn_on_empty_mag_light : BOOL;
    T1_at_end : BOOL;
    extend_mag_slide : BOOL;
    empty_mag_error_solved : BOOL;
    arm_to_home : BOOL;
    retract_mag_slide : BOOL;
    turn_on_vacuum : BOOL;
    turn_off_vacuum : BOOL;
    manual_mode : BOOL;
    set_cycle_end_on : BOOL;
    loop_to_cycle_start : BOOL;
    loop_to_mag_status : BOOL;
END_VAR
VAR_INPUT
    T1_to_end : BOOL;
    T1_to_home : BOOL;
    T1_at_home : BOOL;
    T2_to_end : BOOL;
    T2_to_home : BOOL;
    T2_at_home : BOOL;
    T2_at_end : BOOL;
    vacuum_sensor : BOOL;
END_VAR
VAR_OUTPUT
    vacuum_actuator : BOOL;
END_VAR
VAR_INPUT
    mag_empty : BOOL;
END_VAR
VAR_OUTPUT
    mag_actuator : BOOL;
END_VAR
VAR
    _p1 : BOOL;
    _p2 : BOOL;
    _p3 : BOOL;
END_VAR
(* ladder, written here as Structured Text *)

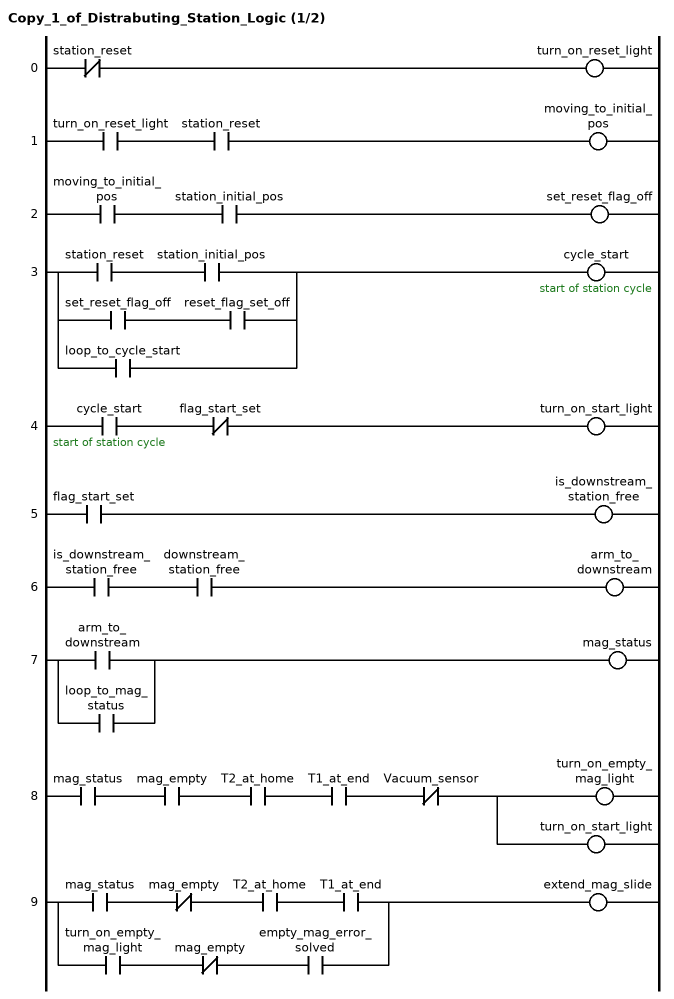
(* Rung 0 *)
turn_on_reset_light := NOT station_reset;
(* Rung 1 *)
moving_to_initial_pos := turn_on_reset_light AND station_reset;
(* Rung 2 *)
set_reset_flag_off := moving_to_initial_pos AND station_initial_pos;
(* Rung 3 *)
cycle_start := (station_reset AND station_initial_pos) OR (set_reset_flag_off AND reset_flag_set_off) OR loop_to_cycle_start;
(* Rung 4 *)
turn_on_start_light := cycle_start AND NOT flag_start_set;
(* Rung 5 *)
is_downstream_station_free := flag_start_set;
(* Rung 6 *)
arm_to_downstream := is_downstream_station_free AND downstream_station_free;
(* Rung 7 *)
mag_status := arm_to_downstream OR loop_to_mag_status;
(* Rung 8 *)
_p1 := mag_status AND mag_empty AND T2_at_home AND T1_at_end AND NOT Vacuum_sensor;
turn_on_empty_mag_light := _p1;
turn_on_start_light := _p1;
(* Rung 9 *)
extend_mag_slide := (mag_status AND NOT mag_empty AND T2_at_home AND T1_at_end) OR (turn_on_empty_mag_light AND NOT mag_empty AND empty_mag_error_solved);

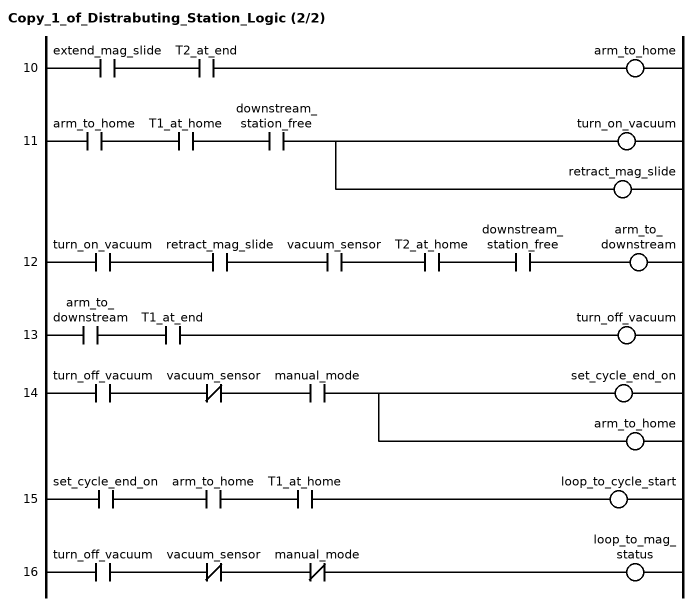
(* Rung 10 *)
arm_to_home := extend_mag_slide AND T2_at_end;
(* Rung 11 *)
_p2 := arm_to_home AND T1_at_home AND downstream_station_free;
turn_on_vacuum := _p2;
retract_mag_slide := _p2;
(* Rung 12 *)
arm_to_downstream := turn_on_vacuum AND retract_mag_slide AND vacuum_sensor AND T2_at_home AND downstream_station_free;
(* Rung 13 *)
turn_off_vacuum := arm_to_downstream AND T1_at_end;
(* Rung 14 *)
_p3 := turn_off_vacuum AND NOT vacuum_sensor AND manual_mode;
set_cycle_end_on := _p3;
arm_to_home := _p3;
(* Rung 15 *)
loop_to_cycle_start := set_cycle_end_on AND arm_to_home AND T1_at_home;
(* Rung 16 *)
loop_to_mag_status := turn_off_vacuum AND NOT vacuum_sensor AND NOT manual_mode;
END_FUNCTION_BLOCK